{attribute 'linkalways'} 
{attribute 'no_explicit_call' := 'This FB is a CLASS and must be accessed using methods or properties'}
{attribute 'enable_dynamic_creation'}
FUNCTION_BLOCK _ETcVnRTrees EXTENDS EnumDatatypeBase
VAR
	localData : ETcVnRTrees;
	activeData : REFERENCE TO ETcVnRTrees;
	enumBaseDatatype : _UDINT(localData);
END_VAR

METHOD PRIVATE AddLocalEnumeration
VAR_INPUT
	Enumeration : T_MAXSTRING;
	Value : ETcVnRTrees;
END_VAR
AddEnumeration(Enumeration, Value);
END_METHOD

PROPERTY PUBLIC Address : PVOID
GET
Address := ADR(activeData);
END_GET
END_PROPERTY

METHOD PUBLIC ClearReference
VAR_INPUT
END_VAR
activeData REF= localData;
SetBaseDatatypeReference();
END_METHOD

METHOD PUBLIC Clone : I_Datatype
VAR
    pClone : POINTER TO _ETcVnRTrees;
END_VAR
pClone := __NEW(_ETcVnRTrees(InitialValue := Value));
Clone := pClone^;
END_METHOD

METHOD FB_init : BOOL
VAR_INPUT
	bInitRetains : BOOL; // if TRUE, the retain variables are initialized (warm start / cold start)
	bInCopyCode : BOOL;  // if TRUE, the instance afterwards gets moved into the copy code (online change)
	InitialValue : ETcVnRTrees;
END_VAR
localData := InitialValue;
AddBaseDatatype(enumBaseDatatype);
ClearReference();

AddLocalEnumeration('TCVN_RT_CLASSIFIER', ETcVnRTrees.TCVN_RT_CLASSIFIER);
AddLocalEnumeration('TCVN_RT_REGRESSOR', ETcVnRTrees.TCVN_RT_REGRESSOR);
END_METHOD

PROPERTY PUBLIC Identifier : T_MAXSTRING
GET
Identifier := 'ETcVnRTrees';
END_GET
END_PROPERTY

METHOD IsEnumeratorValueEqual : BOOL
VAR_INPUT
	Enumerator : I_KeyValueForwardEnumerator;
END_VAR
VAR
	storedValue : ETcVnRTrees;
END_VAR
IF NOT Enumerator.TryGet(storedValue) THEN
	RETURN;
END_IF

IsEnumeratorValueEqual := storedValue = activeData;
END_METHOD

METHOD PUBLIC MakeReferenceTo
VAR_INPUT
	ReferenceTarget : REFERENCE TO ETcVnRTrees;
END_VAR
activeData REF= ReferenceTarget;
SetBaseDatatypeReference();
END_METHOD

METHOD PROTECTED SetBaseDatatypeReference
VAR_INPUT
END_VAR
enumBaseDatatype.MakeReferenceTo(activeData);
END_METHOD

PROPERTY PUBLIC Size : UDINT
GET
Size := SIZEOF(activeData);
END_GET
END_PROPERTY

METHOD TryMakeReferenceTo : BOOL
VAR_INPUT
	Target : I_Datatype;
END_VAR
VAR
	targetAsEnum : I_EnumDatatype;
	pTargetData : POINTER TO ETcVnRTrees;
END_VAR
IF NOT Target.TryResolveAsEnumDatatype(targetAsEnum) THEN
	RETURN;
END_IF

IF targetAsEnum.Identifier <> Identifier THEN
	RETURN;
END_IF

pTargetData := Target.Address;
activeData REF= pTargetData^;
SetBaseDatatypeReference();
TryMakeReferenceTo := TRUE;
END_METHOD

PROPERTY PUBLIC Value : ETcVnRTrees
GET
Value := activeData;
END_GET
SET
activeData := Value;
END_SET
END_PROPERTY

END_FUNCTION_BLOCK

(* stored: Version 1.1.0.1
   POU _ETcVnRTrees: Id {7029f1cb-58d1-4870-8ba6-39006a396bd9}, SpecialFunc None
   Folder Constructor: Id {0cc4a295-386f-4d82-bcac-93b5ce05b62c}
   Folder Private: Id {a34d9b74-711c-445f-b821-dbc81b921d97}
   Folder Protected: Id {d069490d-48ce-457d-b183-669794af5e01}
   Method AddLocalEnumeration: Id {d1ed2f21-7947-4d01-9436-d5783b163290}
   Property Address: Id {b04dce31-2c5d-4576-b480-4b60b1ae813a}
   Get Get: Id {89b6544a-b8e1-4a79-b598-1cdd859e52f4}
   Method ClearReference: Id {e1f17bbc-7fbd-4702-bffd-80edeb78b169}
   Method Clone: Id {b1d127c1-0476-4f0c-bb0b-6cdbe0c05eb7}
   Method FB_init: Id {4858f31d-ba62-4352-92f4-8fb7889c200e}
   Property Identifier: Id {71d723c1-546b-48e5-99d3-7ca235d72ce1}
   Get Get: Id {110fba21-9fb1-4b1e-940f-e6d6d76388ff}
   Method IsEnumeratorValueEqual: Id {d703f31a-980b-4f6e-b9f8-3eb9fc53d3bf}
   Method MakeReferenceTo: Id {bbd9ea8e-2c21-4ae8-8213-585935ced4f7}
   Method SetBaseDatatypeReference: Id {a24f765c-6ec2-4ae2-b85f-52c5dc93fac9}
   Property Size: Id {5f18fe2e-bc8d-4fb0-b89c-8a21e89d92f4}
   Get Get: Id {51c0327b-aaf6-4646-ac6d-cd99a588e96a}
   Method TryMakeReferenceTo: Id {39310a28-d256-4387-82e4-12cb07962abe}
   Property Value: Id {96756f21-f7c3-4bad-825e-f95ec92d96f2}
   Get Get: Id {89a77945-3511-4988-8041-97129ebe00bf}
   Set Set: Id {be8b6ad3-6e3e-4958-879e-aaf7a167ff3e} *)
